{attribute 'qualified_only'}
{attribute 'strict'}
TYPE E_SocketReceiveState :
(
	READY,
	RECEIVING,
	DONE,
	ERROR
);
END_TYPE

(* stored: Version 1.1.0.1, ProductVersion 3.1.4024.13
   DUT E_SocketReceiveState: Id {33916a1f-ceda-4d92-9ced-74fc1680425f} *)
